FUNCTION F_StateEnumToStringGeneralState : String
VAR_INPUT
		eState  : eGeneralState;
END_VAR
VAR
END_VAR

CASE eState OF
	eGeneralState.Idle:
		F_StateEnumToStringGeneralState := 'Idle';
	eGeneralState.Execute:
		F_StateEnumToStringGeneralState := 'Execute';
	eGeneralState.Stopped:
		F_StateEnumToStringGeneralState := 'Stopped';
	eGeneralState.Aborted:
		F_StateEnumToStringGeneralState := 'Aborted';
ELSE
	F_StateEnumToStringGeneralState := 'Unknown';
END_CASE

END_FUNCTION

(* stored: Version 1.1.0.1
   POU F_StateEnumToStringGeneralState: Id {42b1279a-3c78-4fd1-b837-f3a59e245a59}, SpecialFunc None *)
